PROGRAM MAIN
VAR
	FCS :BOOL :=TRUE;
	FCD :BOOL :=FALSE;
	FCA :BOOL :=TRUE;
	FCB :BOOL :=FALSE;
	START :BOOL :=FALSE;
	RESET :BOOL :=FALSE;
	DX :BOOL :=FALSE;
	SX :BOOL :=FALSE;
	SU :BOOL :=FALSE;
	GIU :BOOL :=FALSE;
	ALLARME :BOOL :=FALSE;
END_VAR

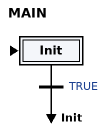
INITIAL_STEP Init:
END_STEP
TRANSITION FROM Init TO Init
    := TRUE;
END_TRANSITION

ACTION ACT3:
GIU :=FALSE;
SU := TRUE;
END_ACTION

ACTION ACT4:
SU :=FALSE;
DX := FALSE;
GIU :=TRUE;
END_ACTION

END_PROGRAM

(* stored: Version 1.1.0.1, ProductVersion 3.1.4024.10
   POU MAIN: Id {f338db10-01d9-496a-b18c-aaf947a63a76}, SpecialFunc None
   Action ACT3: Id {699a5119-e0d8-4a9c-a0b8-bf68060a2a7d}
   Action ACT4: Id {ebe17670-4c8f-4040-bd25-886c2edcc2a6} *)
